{attribute 'qualified_only'}
{attribute 'strict'}
TYPE E_FastDoorState :
(
	INIT,
	CLOSED, 
	OPENING,
	OPEN		
);
END_TYPE

(* stored: Version 1.1.0.1, ProductVersion 3.1.4024.9
   DUT E_FastDoorState: Id {61abd631-1515-4730-b73a-8c1e6e18436f} *)
